// TIA Portal V16 export
// export: Created 2020-03-06T18:52:04.2842381Z, ExportSetting WithDefaults, DisplayName Totally Integrated Automation Portal, DisplayVersion V16, DisplayName TIA Portal Version Control Interface, DisplayVersion V16, DisplayName TIA Portal Openness, DisplayVersion V16, DisplayName TIA Portal Teamcenter Gateway, DisplayVersion V16, DisplayName SINAMICS Startdrive Advanced, DisplayVersion V16 Update 1, DisplayName SINAMICS Startdrive G130, G150, S120, S150, SINAMICS MV, S210, DisplayVersion V16 Update 1, DisplayName SINAMICS Startdrive G110M, G120, G120C, G120D, G120P, DisplayVersion V16 Update 1, DisplayName STEP 7 Professional, DisplayVersion V16, DisplayName STEP 7 Safety, DisplayVersion V16, DisplayName WinCC Professional, DisplayVersion V16
FUNCTION_BLOCK "1oo2 or 2oo2 R"   // FB882, LAD
TITLE = 1oo2 or 2oo2
{ S7_Optimized_Access := 'TRUE' }
VERSION : 0.1
// stored: AutoNumber false, IsIECCheckEnabled false, IsRetainMemResEnabled false, MemoryReserve 100, SetENOAutomatically false, UDAEnableTagReadback false
   VAR_INPUT
      VM : Int;   // Voting Mode - "0=1oo2" "1=2oo2"
      SM : Int;   // Selection Mode - "0=Select Low" "1=Select High"
      V1 : Real;
      V2 : Real;
   END_VAR
   VAR_OUTPUT
      FV : Real;   // Final Value
      LA : Bool;   // Limit Alarm
      GA : Bool;   // General Alarm
   END_VAR
   VAR
      Config : Struct
         GL : Struct   // Global Limits
            HH : Real := 100.0;   // High High
            H : Real := 90.0;   // High
            L : Real := 10.0;   // Low
            LL : Real;   // Low Low
         END_STRUCT;
         H : Real := 1.0;   // Hysteresis
      END_STRUCT;
      V1HHA { ExternalAccessible := 'False'; ExternalVisible := 'False'; ExternalWritable := 'False'} : "HLR";   // Value 1 High High Alarm
      V1HA { ExternalAccessible := 'False'; ExternalVisible := 'False'; ExternalWritable := 'False'} : "HLR";   // Value 1 High Alarm
      V1LA { ExternalAccessible := 'False'; ExternalVisible := 'False'; ExternalWritable := 'False'} : "LLR";   // Value 1 Low Alarm
      V1LLA { ExternalAccessible := 'False'; ExternalVisible := 'False'; ExternalWritable := 'False'} : "LLR";   // Value 1 Low Low Alarm
      V2HHA { ExternalAccessible := 'False'; ExternalVisible := 'False'; ExternalWritable := 'False'} : "HLR";   // Value 2 High High Alarm
      V2HA { ExternalAccessible := 'False'; ExternalVisible := 'False'; ExternalWritable := 'False'} : "HLR";   // Value 2 High Alarm
      V2LA { ExternalAccessible := 'False'; ExternalVisible := 'False'; ExternalWritable := 'False'} : "LLR";   // Value 2 Low Alarm
      V2LLA { ExternalAccessible := 'False'; ExternalVisible := 'False'; ExternalWritable := 'False'} : "LLR";   // Value 2 Low Low Alarm
      SMNV { ExternalAccessible := 'False'; ExternalVisible := 'False'; ExternalWritable := 'False'} : "Min 2R";   // Select Minimum Value
      SMXV { ExternalAccessible := 'False'; ExternalVisible := 'False'; ExternalWritable := 'False'} : "Max 2R";   // Select Maximum Value
   END_VAR
BEGIN

REGION Network 1: V1 High High Alarm
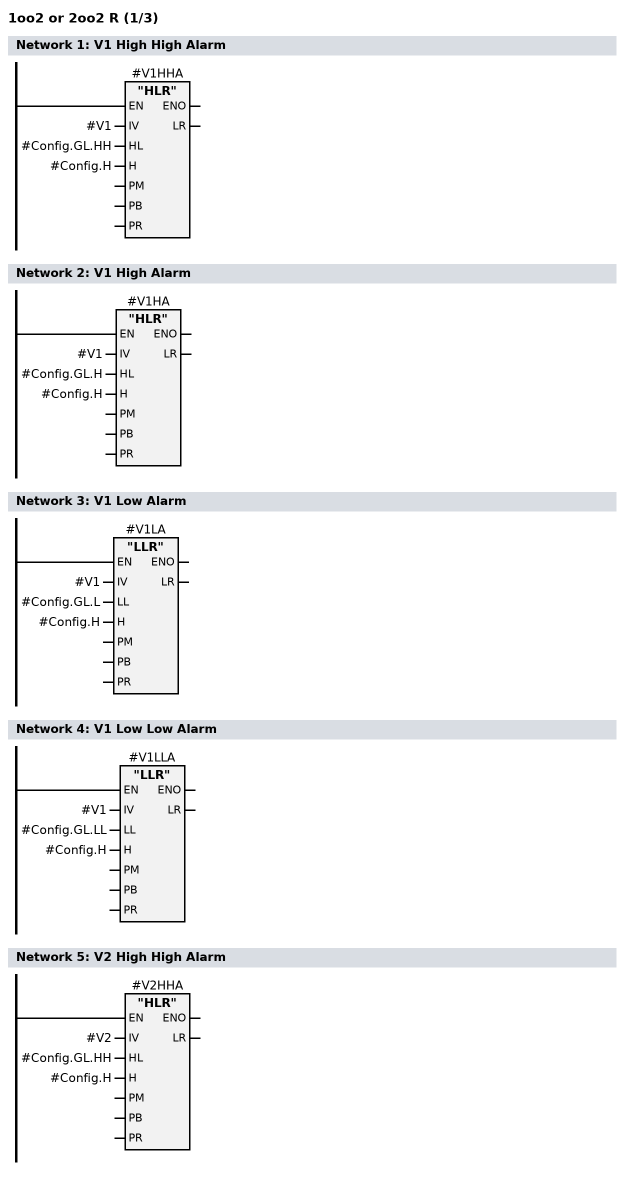
   RUNG wire#powerrail
      #V1HHA(IV := #V1, HL := #Config.GL.HH, H := #Config.H, PM :=, PB :=, PR :=, LR =>)
   END_RUNG
   // the same network as SCL:
   #V1HHA(IV := #V1, HL := #Config.GL.HH, H := #Config.H);   // "HLR"
END_REGION

REGION Network 2: V1 High Alarm
   RUNG wire#powerrail
      #V1HA(IV := #V1, HL := #Config.GL.H, H := #Config.H, PM :=, PB :=, PR :=, LR =>)
   END_RUNG
   // the same network as SCL:
   #V1HA(IV := #V1, HL := #Config.GL.H, H := #Config.H);   // "HLR"
END_REGION

REGION Network 3: V1 Low Alarm
   RUNG wire#powerrail
      #V1LA(IV := #V1, LL := #Config.GL.L, H := #Config.H, PM :=, PB :=, PR :=, LR =>)
   END_RUNG
   // the same network as SCL:
   #V1LA(IV := #V1, LL := #Config.GL.L, H := #Config.H);   // "LLR"
END_REGION

REGION Network 4: V1 Low Low Alarm
   RUNG wire#powerrail
      #V1LLA(IV := #V1, LL := #Config.GL.LL, H := #Config.H, PM :=, PB :=, PR :=, LR =>)
   END_RUNG
   // the same network as SCL:
   #V1LLA(IV := #V1, LL := #Config.GL.LL, H := #Config.H);   // "LLR"
END_REGION

REGION Network 5: V2 High High Alarm
   RUNG wire#powerrail
      #V2HHA(IV := #V2, HL := #Config.GL.HH, H := #Config.H, PM :=, PB :=, PR :=, LR =>)
   END_RUNG
   // the same network as SCL:
   #V2HHA(IV := #V2, HL := #Config.GL.HH, H := #Config.H);   // "HLR"
END_REGION

REGION Network 6: V2 High Alarm
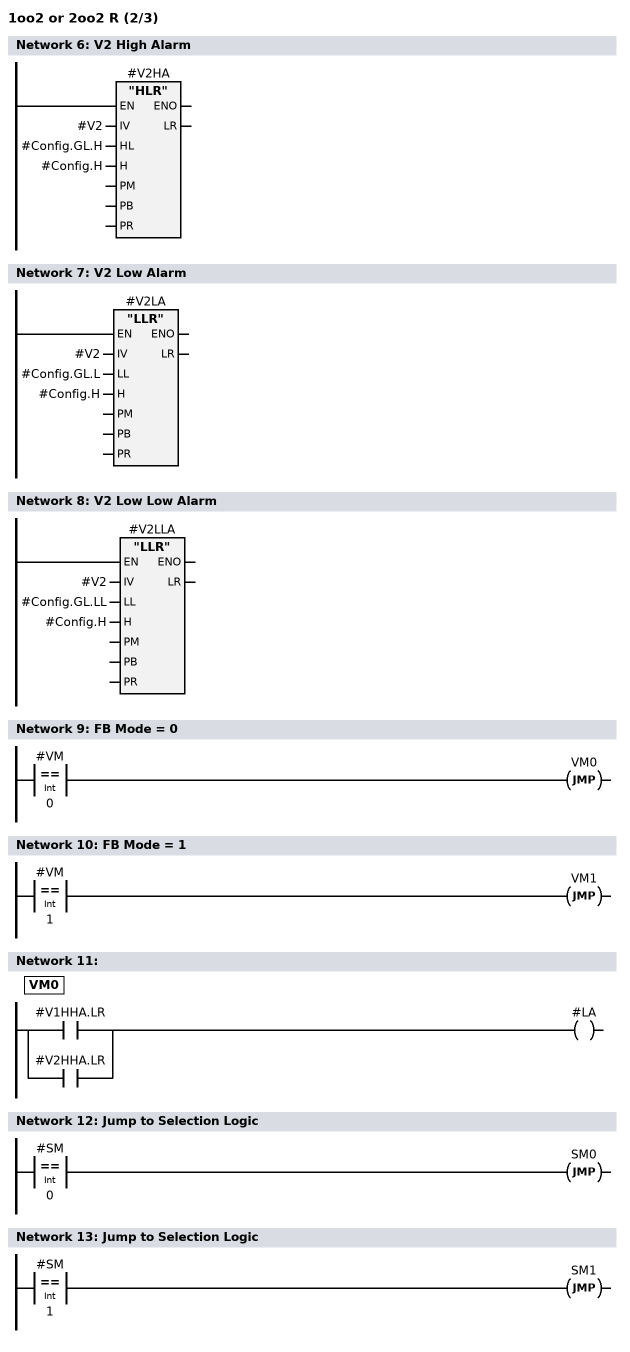
   RUNG wire#powerrail
      #V2HA(IV := #V2, HL := #Config.GL.H, H := #Config.H, PM :=, PB :=, PR :=, LR =>)
   END_RUNG
   // the same network as SCL:
   #V2HA(IV := #V2, HL := #Config.GL.H, H := #Config.H);   // "HLR"
END_REGION

REGION Network 7: V2 Low Alarm
   RUNG wire#powerrail
      #V2LA(IV := #V2, LL := #Config.GL.L, H := #Config.H, PM :=, PB :=, PR :=, LR =>)
   END_RUNG
   // the same network as SCL:
   #V2LA(IV := #V2, LL := #Config.GL.L, H := #Config.H);   // "LLR"
END_REGION

REGION Network 8: V2 Low Low Alarm
   RUNG wire#powerrail
      #V2LLA(IV := #V2, LL := #Config.GL.LL, H := #Config.H, PM :=, PB :=, PR :=, LR =>)
   END_RUNG
   // the same network as SCL:
   #V2LLA(IV := #V2, LL := #Config.GL.LL, H := #Config.H);   // "LLR"
END_REGION

REGION Network 9: FB Mode = 0
   RUNG wire#powerrail
      { S7_Templates := "SrcType := Int" } EQ_Contact(in1 := #VM, in2 := 0)
      JumpCoil( VM0 )
   END_RUNG
   // the same network as SCL:
   IF #VM = 0 THEN GOTO VM0; END_IF;
END_REGION

REGION Network 10: FB Mode = 1
   RUNG wire#powerrail
      { S7_Templates := "SrcType := Int" } EQ_Contact(in1 := #VM, in2 := 1)
      JumpCoil( VM1 )
   END_RUNG
   // the same network as SCL:
   IF #VM = 1 THEN GOTO VM1; END_IF;
END_REGION

REGION Network 11
   Label( VM0 )
   RUNG wire#powerrail
      Contact( #V1HHA.LR )
      wire#w1
      Coil( #LA )
   END_RUNG
   RUNG wire#powerrail
      Contact( #V2HHA.LR )
   END_RUNG wire#w1
   // the same network as SCL:
   VM0:
   #LA := #V1HHA.LR OR #V2HHA.LR;
END_REGION

REGION Network 12: Jump to Selection Logic
   RUNG wire#powerrail
      { S7_Templates := "SrcType := Int" } EQ_Contact(in1 := #SM, in2 := 0)
      JumpCoil( SM0 )
   END_RUNG
   // the same network as SCL:
   IF #SM = 0 THEN GOTO SM0; END_IF;
END_REGION

REGION Network 13: Jump to Selection Logic
   RUNG wire#powerrail
      { S7_Templates := "SrcType := Int" } EQ_Contact(in1 := #SM, in2 := 1)
      JumpCoil( SM1 )
   END_RUNG
   // the same network as SCL:
   IF #SM = 1 THEN GOTO SM1; END_IF;
END_REGION

REGION Network 14
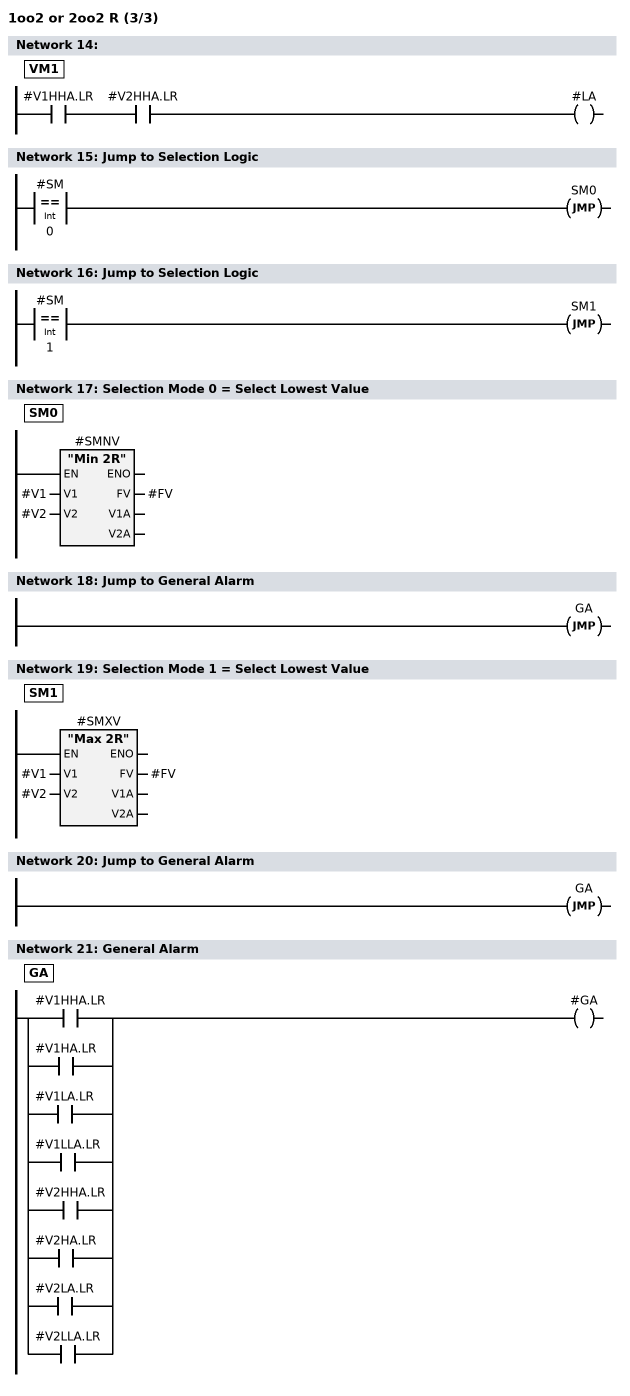
   Label( VM1 )
   RUNG wire#powerrail
      Contact( #V1HHA.LR )
      Contact( #V2HHA.LR )
      Coil( #LA )
   END_RUNG
   // the same network as SCL:
   VM1:
   #LA := #V1HHA.LR AND #V2HHA.LR;
END_REGION

REGION Network 15: Jump to Selection Logic
   RUNG wire#powerrail
      { S7_Templates := "SrcType := Int" } EQ_Contact(in1 := #SM, in2 := 0)
      JumpCoil( SM0 )
   END_RUNG
   // the same network as SCL:
   IF #SM = 0 THEN GOTO SM0; END_IF;
END_REGION

REGION Network 16: Jump to Selection Logic
   RUNG wire#powerrail
      { S7_Templates := "SrcType := Int" } EQ_Contact(in1 := #SM, in2 := 1)
      JumpCoil( SM1 )
   END_RUNG
   // the same network as SCL:
   IF #SM = 1 THEN GOTO SM1; END_IF;
END_REGION

REGION Network 17: Selection Mode 0 = Select Lowest Value
   Label( SM0 )
   RUNG wire#powerrail
      #SMNV(V1 := #V1, V2 := #V2, FV => #FV, V1A =>, V2A =>)
   END_RUNG
   // the same network as SCL:
   SM0:
   #SMNV(V1 := #V1, V2 := #V2, FV => #FV);   // "Min 2R"
END_REGION

REGION Network 18: Jump to General Alarm
   RUNG wire#powerrail
      JumpCoil( GA )
   END_RUNG
   // the same network as SCL:
   GOTO GA;
END_REGION

REGION Network 19: Selection Mode 1 = Select Lowest Value
   Label( SM1 )
   RUNG wire#powerrail
      #SMXV(V1 := #V1, V2 := #V2, FV => #FV, V1A =>, V2A =>)
   END_RUNG
   // the same network as SCL:
   SM1:
   #SMXV(V1 := #V1, V2 := #V2, FV => #FV);   // "Max 2R"
END_REGION

REGION Network 20: Jump to General Alarm
   RUNG wire#powerrail
      JumpCoil( GA )
   END_RUNG
   // the same network as SCL:
   GOTO GA;
END_REGION

REGION Network 21: General Alarm
   Label( GA )
   RUNG wire#powerrail
      Contact( #V1HHA.LR )
      wire#w1
      Coil( #GA )
   END_RUNG
   RUNG wire#powerrail
      Contact( #V1HA.LR )
   END_RUNG wire#w1
   RUNG wire#powerrail
      Contact( #V1LA.LR )
   END_RUNG wire#w1
   RUNG wire#powerrail
      Contact( #V1LLA.LR )
   END_RUNG wire#w1
   RUNG wire#powerrail
      Contact( #V2HHA.LR )
   END_RUNG wire#w1
   RUNG wire#powerrail
      Contact( #V2HA.LR )
   END_RUNG wire#w1
   RUNG wire#powerrail
      Contact( #V2LA.LR )
   END_RUNG wire#w1
   RUNG wire#powerrail
      Contact( #V2LLA.LR )
   END_RUNG wire#w1
   // the same network as SCL:
   GA:
   #GA := #V1HHA.LR OR #V1HA.LR OR #V1LA.LR OR #V1LLA.LR OR #V2HHA.LR OR #V2HA.LR OR #V2LA.LR OR #V2LLA.LR;
END_REGION
END_FUNCTION_BLOCK
